// TwinCAT 3 PLC project Virtual_PLC
// ProgramVersion: 3.1.4024.0
// libraries:
//   Tc2_Standard, * (Beckhoff Automation GmbH)
//   Tc2_System, * (Beckhoff Automation GmbH)
//   Tc3_Module, * (Beckhoff Automation GmbH)
//   VisuSymbols,3.5.10.0,System
// project tree:
//   / GlobalTextList.TcGTLO, PlcTask.TcTTO, Visualization Manager.TcVMO (not stored)
//   GVLs/ GVL.TcGVL
//   POUs/ fbMaking_Coffee.TcPOU, fbMaking_Toast.TcPOU, MAIN.TcPOU
//   VISUs/ Visualization.TcVIS
// real-time tasks:
//   TASK PlcTask: cycle T#10ms, priority 20, ADS port 350

CONFIGURATION Virtual_PLC
    RESOURCE PLC ON TwinCAT3
        TASK PlcTask(INTERVAL := T#10ms, PRIORITY := 20);
        PROGRAM MAIN WITH PlcTask : MAIN;
    END_RESOURCE
END_CONFIGURATION

// ---- GVLs/GVL.TcGVL
{attribute 'qualified_only'}
VAR_GLOBAL

    (* Coffee process *)
	HeatingUp : BOOL;
	ix_Start : BOOL;
	WakeUp : BOOL;
	CoffeeState : INT;
	GrindButton : BOOL;
	CoffeeDone : BOOL;

    (* Breakfast process *)
	InsertedButton : BOOL;
	LeverButton : BOOL;
	ToastState : INT;

    (* Status signals *)
    BreakfastReady : BOOL;
END_VAR

// ---- POUs/MAIN.TcPOU
PROGRAM MAIN
VAR
	MakingCoffee : fbMaking_Coffee;
	MakingToast : fbMaking_Toast;
END_VAR

MakingCoffee(Grinding := GVL.GrindButton, ToastState := GVL.ToastState, GetOffBed := GVL.Wakeup, HeatButton := GVL.HeatingUp, Start := GVL.ix_Start, CoffeeMakingState => GVL.CoffeeState);
MakingToast(LeverDown := GVL.LeverButton, BreadInserted := GVL.InsertedButton, CoffeeState := GVL.CoffeeState, MakingToastState => GVL.ToastState);

END_PROGRAM

// ---- POUs/fbMaking_Coffee.TcPOU
FUNCTION_BLOCK fbMaking_Coffee
VAR_INPUT
	GetOffBed : BOOL;
	HeatButton : BOOL;
	Start : BOOL;
	ToastState : INT;
	Grinding : BOOL;
END_VAR
VAR_OUTPUT
	WaterHeating : BOOL;
	CoffeeMakingState : INT;
END_VAR
VAR
	step: INT;
	WaterHot : BOOL;
	TimerON : TON;
	Brewing : BOOL;
END_VAR

CASE step OF
	0 : // Idle	
		IF GetOffBed = TRUE AND Start THEN
			step := 10;
		END_IF
	10: // Start heating up the water
		IF HeatButton = TRUE THEN
			CoffeeMakingState := 1;
			TimerON(IN := TRUE, PT := T#5S);
		END_IF
		WaterHot := TimerON.Q;
		IF WaterHot = TRUE THEN
			step := 20;
			TimerON(IN := FALSE);
		END_IF
	20 : // Grind the coffee beans
		IF ToastState = 1 AND Grinding THEN
			CoffeeMakingState := 2;
			TimerON(IN := TRUE, PT := T#5S);
		END_IF
		IF TimerON.Q THEN
			step := 30;
			TimerON(IN := FALSE);
		END_IF
	30 : //Brewing the coffee
		IF ToastState = 2 THEN
			Brewing := TRUE;
			CoffeeMakingState := 3;
		END_IF
END_CASE

END_FUNCTION_BLOCK

// ---- POUs/fbMaking_Toast.TcPOU
FUNCTION_BLOCK fbMaking_Toast
VAR_INPUT
	CoffeeState : INT;
	BreadInserted : BOOL;
	LeverDown : BOOL;
END_VAR
VAR
	step : INT;
	Toasting : BOOL;
	TimerON : TON;
	JamDetected: BOOL;
END_VAR
VAR_OUTPUT
	MakingToastState : INT;
END_VAR

CASE step OF
	0 : //Idle
		IF BreadInserted AND CoffeeState = 1 THEN
			step := 10;
		END_IF
	10 : // Loading Bread
		IF LeverDown THEN
			step := 20;
		END_IF
	20 : //Toasting
		IF JamDetected THEN
			step := 0;
		ELSIF NOT JamDetected THEN
			Toasting := TRUE;
			MakingToastState := 1;
		END_IF
		TimerON(IN := Toasting, PT := T#5S);
		IF TimerON.Q THEN
			MakingToastState := 2;
			TimerON(IN := FALSE);
			Making_Toast := TRUE;
		END_IF
END_CASE

END_FUNCTION_BLOCK

// ---- GlobalTextList.TcGTLO
TEXTLIST GlobalTextList
  340 = ' Bread'
  542 = 'Break fast Ready'
  554 = 'Breakfast Ready'
  532 = 'Brewing'
  420 = 'Brewing Done'
  250 = 'Coffee Ready'
  997 = 'Grind Coffee'
  936 = 'GrindingDone'
  789 = 'Heat up water'
  289 = 'Insert'
  928 = 'Insert Bread'
  577 = 'Lever Down'
  278 = 'Making Coffee State: %s'
  196 = 'Making Toast State: %s'
  781 = 'Reset'
  336 = 'Start Coffee'
  469 = 'Toast Error'
  693 = 'Toast Ready'
  127 = 'Wait 5s'
  714 = 'Wake Up'
  930 = 'Water Error'
  15 = 'Water Hot'
END_TEXTLIST

// ---- VISUs/Visualization.TcVIS
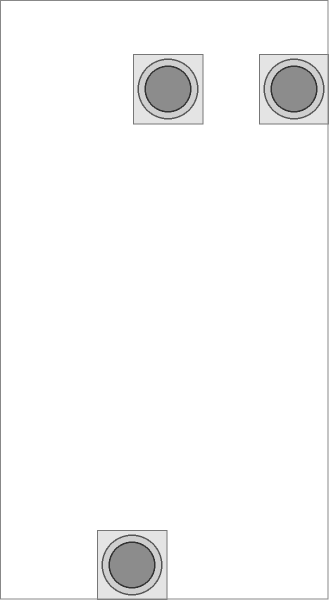
VISUALIZATION Visualization  // 329x600
    PushSwitch (97,530 70x70), behaviour: TOGGLE, style: Switch-PushSwitch-Gray
    PushSwitch (133,54 70x70), variable: GVL.WakeUp, behaviour: TOGGLE, style: Switch-PushSwitch-Gray
    PushSwitch (259,54 70x70), variable: GVL.ix_Start, behaviour: TOGGLE, style: Switch-PushSwitch-Gray
END_VISUALIZATION
